// TIA Portal V18 export
TYPE "MEStoPLC_MainCheckIn_ext"
// stored: IsFailsafeCompliant false
   STRUCT
      Load_Station1PartOK : Bool;   // 订单号
      Load_Station1PartNG : Bool;   // 工件可加工标志位,收到MES.StationReqMesDone后开始加工
      Load_Station1ReqMesDone : Bool;   // 工件可不加工标志位,收到MES.StationReqMesDone后放行
      Load_Station1Spare : Bool;   // Spare
      Load_Station1Spare1 : Bool;   // Spare
      Load_Station1Spare2 : Bool;   // Spare
      Load_Station1Spare3 : Bool;   // Spare
      Load_Station1Spare4 : Bool;   // Spare
      Load_Station2PartOK : Bool;   // 订单号
      Load_Station2PartNG : Bool;   // 工件可加工标志位,收到MES.StationReqMesDone后开始加工
      Load_Station2ReqMesDone : Bool;   // 工件可不加工标志位,收到MES.StationReqMesDone后放行
      Load_Station2Spare : Bool;   // Spare
      Load_Station2Spare1 : Bool;   // Spare
      Load_Station2Spare2 : Bool;   // Spare
      Load_Station2Spare3 : Bool;   // Spare
      Load_Station2Spare4 : Bool;   // Spare
      Load_Station3PartOK : Bool;   // 订单号
      Load_Station3PartNG : Bool;   // 工件可加工标志位,收到MES.StationReqMesDone后开始加工
      Load_Station3ReqMesDone : Bool;   // 工件可不加工标志位,收到MES.StationReqMesDone后放行
      Load_Station3Spare : Bool;   // Spare
      Load_Station3Spare1 : Bool;   // Spare
      Load_Station3Spare2 : Bool;   // Spare
      Load_Station3Spare3 : Bool;   // Spare
      Load_Station3Spare4 : Bool;   // Spare
      Load_Station4PartOK : Bool;   // 订单号
      Load_Station4PartNG : Bool;   // 工件可加工标志位,收到MES.StationReqMesDone后开始加工
      Load_Station4ReqMesDone : Bool;   // 工件可不加工标志位,收到MES.StationReqMesDone后放行
      Load_Station4Spare : Bool;   // Spare
      Load_Station4Spare1 : Bool;   // Spare
      Load_Station4Spare2 : Bool;   // Spare
      Load_Station4Spare3 : Bool;   // Spare
      Load_Station4Spare4 : Bool;   // Spare
      Load_Station5PartOK : Bool;   // 订单号
      Load_Station5PartNG : Bool;   // 工件可加工标志位,收到MES.StationReqMesDone后开始加工
      Load_Station5ReqMesDone : Bool;   // 工件可不加工标志位,收到MES.StationReqMesDone后放行
      Load_Station5Spare : Bool;   // Spare
      Load_Station5Spare1 : Bool;   // Spare
      Load_Station5Spare2 : Bool;   // Spare
      Load_Station5Spare3 : Bool;   // Spare
      Load_Station5Spare4 : Bool;   // Spare
      Load_Station6PartOK : Bool;   // 订单号
      Load_Station6PartNG : Bool;   // 工件可加工标志位,收到MES.StationReqMesDone后开始加工
      Load_Station6ReqMesDone : Bool;   // 工件可不加工标志位,收到MES.StationReqMesDone后放行
      Load_Station6Spare : Bool;   // Spare
      Load_Station6Spare1 : Bool;   // Spare
      Load_Station6Spare2 : Bool;   // Spare
      Load_Station6Spare3 : Bool;   // Spare
      Load_Station6Spare4 : Bool;   // Spare
      Load_Station7PartOK : Bool;   // 订单号
      Load_Station7PartNG : Bool;   // 工件可加工标志位,收到MES.StationReqMesDone后开始加工
      Load_Station7ReqMesDone : Bool;   // 工件可不加工标志位,收到MES.StationReqMesDone后放行
      Load_Station7Spare : Bool;   // Spare
      Load_Station7Spare1 : Bool;   // Spare
      Load_Station7Spare2 : Bool;   // Spare
      Load_Station7Spare3 : Bool;   // Spare
      Load_Station7Spare4 : Bool;   // Spare
      Load_Station8PartOK : Bool;   // 订单号
      Load_Station8PartNG : Bool;   // 工件可加工标志位,收到MES.StationReqMesDone后开始加工
      Load_Station8ReqMesDone : Bool;   // 工件可不加工标志位,收到MES.StationReqMesDone后放行
      Load_Station8Spare : Bool;   // Spare
      Load_Station8Spare5 : Bool;   // Spare
      Load_Station8Spare6 : Bool;   // Spare
      Load_Station8Spare8 : Bool;   // Spare
      Load_Station8Spare9 : Bool;   // Spare
   END_STRUCT;
END_TYPE
